{attribute 'qualified_only'}
{attribute 'strict'}
TYPE eConditionCheck :
(
	INIT := 0,
	READY := 1,
	ERROR := 2,
	SLEEP := 3
);
END_TYPE

(* stored: Version 1.1.0.1, ProductVersion 3.1.4024.12
   DUT eConditionCheck: Id {dcaebc43-7ee5-463b-bf6d-8ef9d0a436df} *)
